function_block abstract FB_Syntax_AbstractBase implements I_Syntax_Widget
var
    _nBaseId : dint;
    _bReady : bool;
end_var

method abstract M_GetValue : int
END_METHOD

method M_Init : bool
M_Init := TRUE;
END_METHOD

method abstract M_Reset : bool
END_METHOD

property P_Name : string
GET
var
end_var
P_Name := 'Base';
END_GET
END_PROPERTY

property P_Ready : bool
GET
var
end_var
P_Ready := _bReady;
END_GET
END_PROPERTY

END_FUNCTION_BLOCK

(* stored: Version 1.1.0.1, ProductVersion 3.1.4024.16
   POU FB_Syntax_AbstractBase: Id {22e123ae-c20b-4e1c-aef1-d6fd464b5691}, SpecialFunc None
   Method M_GetValue: Id {78409f0b-e366-4d15-9455-6f500c60c8d8}
   Method M_Init: Id {5899f78d-24ab-4969-b34b-894490a47980}
   Method M_Reset: Id {a1b2c3d4-e5f6-4a1b-8c2d-3e4f5a6b7c8d}
   Property P_Name: Id {2154926d-de2c-40ee-a734-5322b86599f2}
   Get Get: Id {53c63b8c-93ba-46e3-aa7b-f567464634ad}
   Property P_Ready: Id {b2c3d4e5-f6a1-4b2c-9d3e-4f5a6b7c8d9e}
   Get Get: Id {c3d4e5f6-a1b2-4c3d-ae4f-5a6b7c8d9e0f} *)
